DATA_BLOCK DB 210
VERSION : 0.1
  STRUCT
   ID_Ricetta : INT ;
   PartNumber : ARRAY  [0 .. 31 ] OF //Part number in lavorazione
   CHAR ;
   ToolType : INT ;	//Tool type
   ToolCode : INT ;	//Codice su attrezzo - ingressi digitali
   Anello1Abilitato : BOOL ;
   Anello2Abilitato : BOOL ;
   Velocita_asse_X1 : DINT ;
   Velocita_asse_Y1 : DINT ;
   spare48 : DINT ;
   spare52 : DINT ;
   spare56 : DINT ;
   spare60 : DINT ;
   spare64 : DINT ;
   spare68 : DINT ;
   spare72 : DINT ;
   spare76 : INT ;
   Disable : STRUCT 	//da indirizzo 78
    CkCodicePortapezzo : BOOL ;
    CkPresAnelloAdattamento : BOOL ;
    CkPresenzaNozzleRing : BOOL ;
    CkPresenzaPipe : BOOL ;
    CheckSpare4 : BOOL ;
    CheckSpare5 : BOOL ;
    CheckSpare6 : BOOL ;
    CheckSpare7 : BOOL ;
    CheckSpare8 : BOOL ;
    CheckSpare9 : BOOL ;
   END_STRUCT ;
   NumeroPosizioni : INT ;
   posizioni : ARRAY  [0 .. 19 ] OF //da indirizzo 82
   STRUCT
    X : DINT ;	//1/100 mm
    Y : DINT ;	//1/100 mm
    TempoRibaditura : DINT ;	//msec
   END_STRUCT ;
   spare : ARRAY  [0 .. 38 ] OF INT ;
  END_STRUCT ;	
BEGIN
   ID_Ricetta := 1;
   PartNumber[0] := 'R';
   PartNumber[1] := 'P';
   PartNumber[2] := 'V';
   PartNumber[3] := 'O';
   PartNumber[4] := ' ';
   PartNumber[5] := 'A';
   PartNumber[6] := 'P';
   PartNumber[7] := 'O';
   PartNumber[8] := '0';
   PartNumber[9] := '4';
   PartNumber[10] := ' ';
   PartNumber[11] := ' ';
   PartNumber[12] := ' ';
   PartNumber[13] := ' ';
   PartNumber[14] := ' ';
   PartNumber[15] := ' ';
   PartNumber[16] := ' ';
   PartNumber[17] := ' ';
   PartNumber[18] := ' ';
   PartNumber[19] := ' ';
   PartNumber[20] := ' ';
   PartNumber[21] := ' ';
   PartNumber[22] := ' ';
   PartNumber[23] := ' ';
   PartNumber[24] := ' ';
   PartNumber[25] := ' ';
   PartNumber[26] := ' ';
   PartNumber[27] := ' ';
   PartNumber[28] := ' ';
   PartNumber[29] := ' ';
   PartNumber[30] := ' ';
   PartNumber[31] := ' ';
   ToolType := 1;
   ToolCode := 3;
   Anello2Abilitato := TRUE;
   Velocita_asse_X1 := L#100000;
   Velocita_asse_Y1 := L#100000;
   NumeroPosizioni := 3;
   posizioni[0].X := L#-24040;
   posizioni[0].Y := L#-24040;
   posizioni[0].TempoRibaditura := L#3000;
   posizioni[1].X := L#30290;
   posizioni[1].Y := L#-15440;
   posizioni[1].TempoRibaditura := L#3000;
   posizioni[2].X := L#5320;
   posizioni[2].Y := L#33580;
   posizioni[2].TempoRibaditura := L#3000;
END_DATA_BLOCK

DATA_BLOCK DB 220
VERSION : 0.1
  STRUCT
   General : UDT 200;
   Restore : UDT 200;
  END_STRUCT ;	
BEGIN
// 44 bytes; values not shown
END_DATA_BLOCK

DATA_BLOCK DB 400
VERSION : 0.0
FB 102
BEGIN
END_DATA_BLOCK

DATA_BLOCK DB 401
VERSION : 0.0
FB 102
BEGIN
END_DATA_BLOCK

DATA_BLOCK DB 402
VERSION : 0.0
FB 102
BEGIN
END_DATA_BLOCK

DATA_BLOCK DB 403
VERSION : 0.0
FB 102
BEGIN
END_DATA_BLOCK

DATA_BLOCK DB 404
VERSION : 0.0
FB 102
BEGIN
END_DATA_BLOCK

DATA_BLOCK DB 405
VERSION : 0.0
FB 102
BEGIN
END_DATA_BLOCK

DATA_BLOCK DB 406
VERSION : 0.0
FB 102
BEGIN
END_DATA_BLOCK

DATA_BLOCK DB 407
VERSION : 0.0
FB 102
BEGIN
END_DATA_BLOCK

DATA_BLOCK DB 420
AUTHOR : Castel
VERSION : 0.0
FB 450
BEGIN
END_DATA_BLOCK

DATA_BLOCK DB 421
AUTHOR : Castel
VERSION : 0.0
FB 450
BEGIN
END_DATA_BLOCK

DATA_BLOCK DB 425
VERSION : 0.0
FB 455
BEGIN
END_DATA_BLOCK

DATA_BLOCK DB 426
VERSION : 0.0
FB 455
BEGIN
END_DATA_BLOCK

DATA_BLOCK DB 430
VERSION : 0.0
FB 120
BEGIN
END_DATA_BLOCK

DATA_BLOCK DB 431
VERSION : 0.0
FB 121
BEGIN
END_DATA_BLOCK

DATA_BLOCK DB 435
VERSION : 0.0
FB 221
BEGIN
END_DATA_BLOCK

DATA_BLOCK DB 436
VERSION : 0.0
FB 220
BEGIN
END_DATA_BLOCK

DATA_BLOCK DB 437
VERSION : 0.0
FB 171
BEGIN
END_DATA_BLOCK

DATA_BLOCK DB 438
VERSION : 0.0
FB 170
BEGIN
END_DATA_BLOCK

DATA_BLOCK DB 440
VERSION : 0.0
FB 60
BEGIN
END_DATA_BLOCK

ORGANIZATION_BLOCK OB 1
TITLE = "Main Program Sweep (Cycle)"
VERSION : 0.1
VAR_TEMP
  OB1_EV_CLASS : BYTE ;	//Bits 0-3 = 1 (Coming event), Bits 4-7 = 1 (Event class 1)
  OB1_SCAN_1 : BYTE ;	//1 (Cold restart scan 1 of OB 1), 3 (Scan 2-n of OB 1)
  OB1_PRIORITY : BYTE ;	//Priority of OB Execution
  OB1_OB_NUMBR : BYTE ;	//1 (Organization block 1, OB1)
  OB1_RESERVED_1 : BYTE ;	//Reserved for system
  OB1_RESERVED_2 : BYTE ;	//Reserved for system
  OB1_PREV_CYCLE : INT ;	//Cycle time of previous OB1 scan (milliseconds)
  OB1_MIN_CYCLE : INT ;	//Minimum cycle time of OB1 (milliseconds)
  OB1_MAX_CYCLE : INT ;	//Maximum cycle time of OB1 (milliseconds)
  OB1_DATE_TIME : DATE_AND_TIME ;	//Date and time OB1 started
END_VAR
BEGIN
NETWORK
TITLE = Bit Alw_ON e ALW_OFF
      SET;
      =     M 100.0;
      NOT;
      =     M 100.1;
NETWORK
TITLE = Line
      CALL  FC 50;
NETWORK
TITLE = OP10
      CALL  FC 100;
NETWORK
TITLE = OP20
      CALL  FC 150;
NETWORK
TITLE = op40
      CALL  FC 200;
NETWORK
TITLE =
NETWORK
TITLE = Reset first scan
      CLR;
      =     M 100.2;
END_ORGANIZATION_BLOCK
